FUNCTION_BLOCK DataPanel_xDB0808_DIO_SAE_J1939 (* Service Interface Function Block Type *)
  (* Standard: SAE J1939; Function: Combo Block: 8 Inputs/8 Outputs (includes all input/output types); Type: DP-34044-1-000 *)
  (* Version 1.0, 2018-12-05, Jose Cabral *)
  (* Version 1.0, 2022-08-04, Franz Höpfinger, Unknown *)
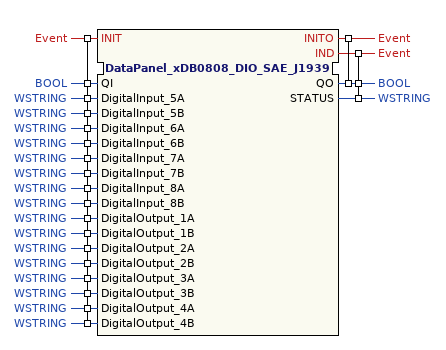
  EVENT_INPUT
    INIT WITH DigitalInput_5A, DigitalInput_5B, DigitalInput_7A, DigitalInput_6A, DigitalInput_6B, DigitalInput_7B, DigitalInput_8A, DigitalInput_8B, DigitalOutput_1A, DigitalOutput_1B, DigitalOutput_3A, DigitalOutput_2A, DigitalOutput_2B, DigitalOutput_3B, DigitalOutput_4A, DigitalOutput_4B, QI; (* Service Initialization *)
  END_EVENT
  EVENT_OUTPUT
    INITO WITH QO; (* Initialization Confirm *)
    IND WITH QO, STATUS; (* Indication from Resource *)
  END_EVENT
  VAR_INPUT
    QI : BOOL; (* Event Input Qualifier *)
    DigitalInput_5A : WSTRING;
    DigitalInput_5B : WSTRING;
    DigitalInput_6A : WSTRING;
    DigitalInput_6B : WSTRING;
    DigitalInput_7A : WSTRING;
    DigitalInput_7B : WSTRING;
    DigitalInput_8A : WSTRING;
    DigitalInput_8B : WSTRING;
    DigitalOutput_1A : WSTRING;
    DigitalOutput_1B : WSTRING;
    DigitalOutput_2A : WSTRING;
    DigitalOutput_2B : WSTRING;
    DigitalOutput_3A : WSTRING;
    DigitalOutput_3B : WSTRING;
    DigitalOutput_4A : WSTRING;
    DigitalOutput_4B : WSTRING;
  END_VAR
  VAR_OUTPUT
    QO : BOOL; (* Event Output Qualifier *)
    STATUS : WSTRING; (* Service Status *)
  END_VAR
END_FUNCTION_BLOCK
